FUNCTION_BLOCK FB_Child EXTENDS FB_Base IMPLEMENTS I_Interface, I_Interface2
VAR
	SomeText : STRING;
	Counter : DINT := 1;
	Result : DINT := 2;
	
	Base : FB_Base;
END_VAR

SomeText:= 'Current counts';

IF Conditions[1] AND Conditions[2]  AND Conditions[3] AND Conditions[4] AND Conditions[5]AND Conditions[6] THEN
	Counter :=Counter+ 1;

	IF Counter > 2 THEN
	Counter := Counter + 5 ;
	END_IF
END_IF

Base(Variable1:=2, Variable2:=3 , Variable3:= 5,Sentence:='', Conditions :=Conditions);


AddTwoInts(    Variable1 :=4,
    Variable2:=4);

METHOD AddTwoInts : DINT
VAR_INPUT
	Variable1 : DINT;
	Variable2 : DINT;
END_VAR
AddTwoInts:=Variable1+Variable2 ;
END_METHOD

PROPERTY PRIVATE AnotherProperty : LREAL
GET
VAR
	percent : LREAL := 100;
END_VAR
END_GET
SET
VAR
	sName : STRING(20) := 'This is the one!';
END_VAR
END_SET
END_PROPERTY

PROPERTY Counted : DINT
GET
VAR
	AddOne : DINT := 1;
END_VAR
END_GET
SET
VAR
	SubTractTwo : DINT := 2;
END_VAR
END_SET
END_PROPERTY

METHOD SecondMethod : BOOL
VAR_INPUT
	bBool : BOOL;
END_VAR
END_METHOD

END_FUNCTION_BLOCK

(* stored: Version 1.1.0.1, ProductVersion 3.1.4024.3
   POU FB_Child: Id {16c60171-46ae-4c0f-982d-d26906c8a65a}, SpecialFunc None
   Method AddTwoInts: Id {6a4e1f8c-f7f9-4983-b9b4-e06e406d35d9}
   Property AnotherProperty: Id {aa0cfd4f-5e29-4982-9f71-257c1439d0f2}
   Get Get: Id {d44792da-1b4d-4983-85ab-83fe99d160dd}
   Set Set: Id {39df90cf-cdb1-4cd9-b65e-5832b944cb70}
   Property Counter: Id {d49735b6-a4d9-4d67-adc2-f3998b3471ec}
   Get Get: Id {7c33609a-907f-4f05-8aea-95e3f6a224e3}
   Set Set: Id {4bb13cca-2444-4335-a94c-c714ed95062a}
   Method SecondMethod: Id {f5bbaa77-a784-4d59-b884-5b52362ac1cd} *)
